Universal Robots URScript: move_modified.script

def move_to_center():
  global _hidden_verificationVariable=0
  set_tool_communication(False, 115200, 0, 1, 1.5, 3.5)
  set_tool_output_mode(0)
  set_tool_digital_output_mode(0, 1)
  set_tool_digital_output_mode(1, 1)
  set_tool_voltage(0)
  set_safety_mode_transition_hardness(1)
  set_standard_analog_input_domain(0, 1)
  set_standard_analog_input_domain(1, 1)
  set_tool_analog_input_domain(0, 1)
  set_tool_analog_input_domain(1, 1)
  set_analog_outputdomain(0, 0)
  set_analog_outputdomain(1, 0)
  set_input_actions_to_default()
  set_target_payload(0.530000, [0.009000, -0.039000, 0.092000], [0.000534, 0.000534, 0.000534, 0.000000, 0.000000, 0.000000])
  set_tcp(p[0.0,0.0,0.11,0.0,0.0,0.0])
  set_gravity([0.0, 0.0, 9.82])
  global Al_plate=p[0.12405209206180495,-0.2666666051843552,0.020008101224669964,-9.276623980477388E-5,1.8107917580596192E-5,3.1233857134705927]
  global Frame2x2=p[0.18266245434305164,-0.34273121659514855,0.026002571110600767,-2.225423529876215E-4,3.0110667546023537E-4,3.1233976058306383]
  global URlogoTutorial=p[-0.08178353973148575,-0.3363174165299142,0.04788621506469384,-3.9746155723688456E-5,-3.4682148779121894E-5,-1.5668291789091222]
  global carouselrod=p[0.2020731702281844,-0.34951442511341274,0.1947611446273096,3.139766958234101,-0.10689428010274801,-1.1796370330365635E-5]
  global paper=p[-0.09670794781244417,-0.3283412964648025,0.027665994240809913,-3.2057893450593004E-5,2.867088716161181E-5,-1.6085327915291054]
  global rod=p[0.13368013097420872,-0.41123185103490206,0.09926814901395645,2.2214229924093103,-2.2214158162465862,-2.9165882738638143E-5]
  # begin: URCap Installation Node
  global c1_p=p[0.09566676089273368, -0.27623557885180994, 20.0, 0, 3.14159, 0]
  global c2_p=p[0.09567610847471325, -0.25422453802926603, 20.0, 0, 3.14159, 0]
  global c3_p=p[0.07665092863509039, -0.2871041162314084, 20.0, 0, 3.14159, 0]
  global c4_p=p[0.0765982791385102, -0.26510758446858584, 20.0, 0, 3.14159, 0]
  global c5_p=p[0.07661492338844747, -0.2432293411076338, 20.0, 0, 3.14159, 0]
  global c6_p=p[0.05767608239841023, -0.2761239127299706, 20.0, 0, 3.14159, 0]
  global c7_p=p[0.05763317163738289, -0.25406828079349253, 20.0, 0, 3.14159, 0]
  global c1_q=[1.5281997168255637, -1.6486971446621759, 1.6123511746145105, -1.5344503567472312, -1.5707963267948966, 1.5281997168255637]
  global c2_q=[1.5236208569423668, -1.741846715617347, 1.692245110752121, -1.5211947219296706, -1.5707963267948966, 1.5236208569423668]
  global c3_q=[1.5198887450487801, -1.8335093851517774, 1.761278062745017, -1.4985650043881362, -1.5707963267948966, 1.5198887450487801]
  global c4_q=[1.4539822336394537, -1.7199155934021537, 1.6743231027089642, -1.525203836101707, -1.5707963267948966, 1.4539822336394537]
  global c5_q=[1.4434107276785597, -1.816740250633318, 1.749353755032525, -1.5034098311941038, -1.5707963267948966, 1.4434107276785597]
  global c6_q=[0.38325737973488283, -2.3257758095425167, 1.974470662814782, -1.2194911800671617, -1.5707963267948966, 0.38325737973488283]
  global c7_q=[0.4736275351764019, -2.364179239792936, 1.979913771856397, -1.1865308588583574, -1.5707963267948966, 0.4736275351764019]
  global c8_q=[0.8048397284577823, -2.3337203701363913, 1.9757368048081096, -1.2128127614666149, -1.5707963267948966, 0.8048397284577823]
  global c9_q=[0.7905131984043816, -2.3155485561474443, 1.9727344015267305, -1.2279821721741828, -1.5707963267948966, 0.7905131984043816]
  global c10_q=[1.2595250603655543, -1.402133970827033, 1.3529953557654222, -1.5216577117332857, -1.5707963267948966, 1.2595250603655543]
  global c11_q=[1.1244612242815093, -1.8557284430729934, 1.7765947025837907, -1.4916625863056938, -1.5707963267948966, 1.1244612242815093]
  global c12_q=[1.215094687502614, -1.612803849492599, 1.578922938480139, -1.5369154157824367, -1.5707963267948966, 1.215094687502614]
  #   Source: External Control, 1.0.5, FZI Research Center for Information Technology
  #   Type: External Control
  # end: URCap Installation Node
  step_count_c0b60bdf_8f3b_4db0_b670_6f220ad7429b = 0.0
  thread Step_Counter_Thread_9e4d85a9_1c70_45fe_9fb9_d5c392e96989():
    while (True):
      step_count_c0b60bdf_8f3b_4db0_b670_6f220ad7429b = step_count_c0b60bdf_8f3b_4db0_b670_6f220ad7429b + 1.0
      sync()
    end
  end
  run Step_Counter_Thread_9e4d85a9_1c70_45fe_9fb9_d5c392e96989()

  $ 2 "Robot Program"
  $ 3 "MoveJ"
  $ 4 "c1" "breakAfter"
  movel(c1_q, a=0.37, v=0.25)
    movel(c2_q,a=0.37, v=0.27)
    movel(c3_q, a=0.37, v=0.27)
    movel(c4_q, a=0.37, v=0.27)
    movel(c5_q, a=0.37, v=0.27)
    movel(c6_q, a=0.37, v=0.27)
    movel(c7_q, a=0.37, v=0.27)
end
